FUNCTION_BLOCK FB_HeatingSystem
VAR_INPUT
	bEnable : BOOL;
	bExecute : BOOL;
	
	nMaxTemp : UINT;
	nTemp : UINT;
END_VAR
VAR_OUTPUT
	bVentilator1 : BOOL;
	bVentilator2 : BOOL;
	bVentilator3 : BOOL;
	nHeizpatrone : UINT := 0;

	eStatus : State := State.Off;
END_VAR
VAR
	nHeat : REAL := 0;
	timer : TON;
	timer1 : TON;
	eState : StateHeat := StateHeat.Off;
END_VAR

nHeizpatrone := TO_UINT(F_map(nHeat, 0, 5, 0, 16383));

IF NOT bEnable THEN
	eState:= StateHeat.Off;
END_IF

CASE eState OF
StateHeat.Off:
	eStatus := State.Off;
	
	bVentilator1 := FALSE;
	bVentilator2 := FALSE;
	bVentilator3 := FALSE;
	nHeat := 0;
	
	IF bEnable THEN
		eState := StateHeat.Init;
	END_IF
	
StateHeat.Init:
	eStatus := State.Busy;
	bVentilator1 := TRUE;
	bVentilator2 := TRUE;
	bVentilator3 := TRUE;
	
	IF nTemp <= nMaxTemp THEN
		eState := StateHeat.Ready;
	END_IF

StateHeat.Ready:
	eStatus := State.Ready;
	
	nHeat := 0;
	
	IF bExecute THEN
		eState := StateHeat.Heat;
	END_IF

StateHeat.Heat:
	eStatus := State.Busy;
	
	nHeat := 5;
	
	IF nTemp >= 3000 THEN
		nHeat := 0;
		eState := StateHeat.Hold;
	END_IF
	
StateHeat.Hold:
	eStatus := State.Busy;
	
	timer(IN := TRUE, PT := T#30S);
	
	IF nTemp >= 3700 THEN
		nHeat := 0;
	ELSIF nTemp <= 3500 THEN
		timer1(IN := TRUE, PT:= T#500MS);
		IF timer1.Q THEN
			timer1(IN := FALSE);
			nHeat := nHeat + 0.05;
			IF nHeat >= 5 THEN
				nHeat := 5;
			END_IF
		END_IF	

	END_IF
	
	IF timer.Q THEN
		timer(IN := FALSE);
		nHeat := 0;
		eState := StateHeat.Done;
	END_IF	

StateHeat.Done:
	eStatus := State.Done;
	
	nHeat := 0;
	
	IF NOT bExecute THEN
		eState := StateHeat.Init;
	END_IF
	
END_CASE

END_FUNCTION_BLOCK

(* stored: Version 1.1.0.1, ProductVersion 3.1.4024.6
   POU FB_HeatingSystem: Id {7c7b126e-8b79-4d92-8382-02f37357639c}, SpecialFunc None *)
